% RSLogix 500 project Blue Banner Restacker.RSS, saved by version 11.00.00.00 %
PROJECT "UNTITLED"    % processor: MicroLogix 1400 %

PROGRAM FILES
  LAD 2   20 rungs

DATA FILES
  O0 OUTPUT  6 elements
  I1 INPUT  8 elements
  S2 STATUS  66 elements
  B3 BINARY  2 elements
  T4 TIMER  1 elements
  C5 COUNTER  1 elements
  R6 CONTROL  1 elements
  N7 INTEGER  1 elements
  F8 FLOAT  1 elements

LADDER 2
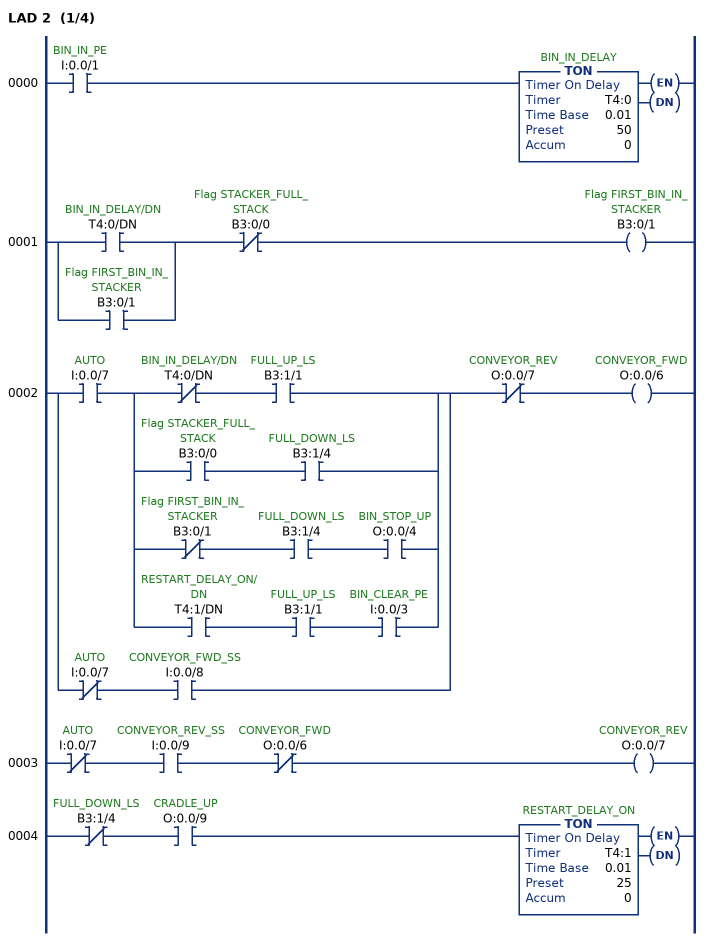
% Rung: 0 %  % edit flag set %
SOR XIC I:0.0/1 TON T4:0 0.01 50 0 EOR
%   I:0.0/1  BIN_IN_PE %
%   T4:0  BIN_IN_DELAY %
% Rung: 1 %  % edit flag set %
SOR BST XIC T4:0/DN NXB XIC B3:0/1 BND XIO B3:0/0 OTE B3:0/1 EOR
%   T4:0  BIN_IN_DELAY %
%   B3:0/1  FIRST_BIN_IN_STACKER  "Flag" %
%   B3:0/0  STACKER_FULL_STACK  "Flag" %
% Rung: 2 %  % edit flag set %
SOR BST XIC I:0.0/7 BST XIO T4:0/DN XIC B3:1/1 NXB BST XIC B3:0/0 XIC B3:1/4 NXB BST XIO B3:0/1 XIC B3:1/4 XIC O:0.0/4 NXB XIC T4:1/DN XIC B3:1/1 XIC I:0.0/3 BND BND BND NXB XIO I:0.0/7 XIC I:0.0/8 BND XIO O:0.0/7 OTE O:0.0/6 EOR
%   I:0.0/7  AUTO %
%   T4:0  BIN_IN_DELAY %
%   B3:1/1  FULL_UP_LS %
%   B3:0/0  STACKER_FULL_STACK  "Flag" %
%   B3:1/4  FULL_DOWN_LS %
%   B3:0/1  FIRST_BIN_IN_STACKER  "Flag" %
%   O:0.0/4  BIN_STOP_UP %
%   T4:1  RESTART_DELAY_ON %
%   I:0.0/3  BIN_CLEAR_PE %
%   I:0.0/8  CONVEYOR_FWD_SS %
%   O:0.0/7  CONVEYOR_REV %
%   O:0.0/6  CONVEYOR_FWD %
% Rung: 3 %  % edit flag set %
SOR XIO I:0.0/7 XIC I:0.0/9 XIO O:0.0/6 OTE O:0.0/7 EOR
%   I:0.0/7  AUTO %
%   I:0.0/9  CONVEYOR_REV_SS %
%   O:0.0/6  CONVEYOR_FWD %
%   O:0.0/7  CONVEYOR_REV %
% Rung: 4 %  % edit flag set %
SOR XIO B3:1/4 XIC O:0.0/9 TON T4:1 0.01 25 0 EOR
%   B3:1/4  FULL_DOWN_LS %
%   O:0.0/9  CRADLE_UP %
%   T4:1  RESTART_DELAY_ON %

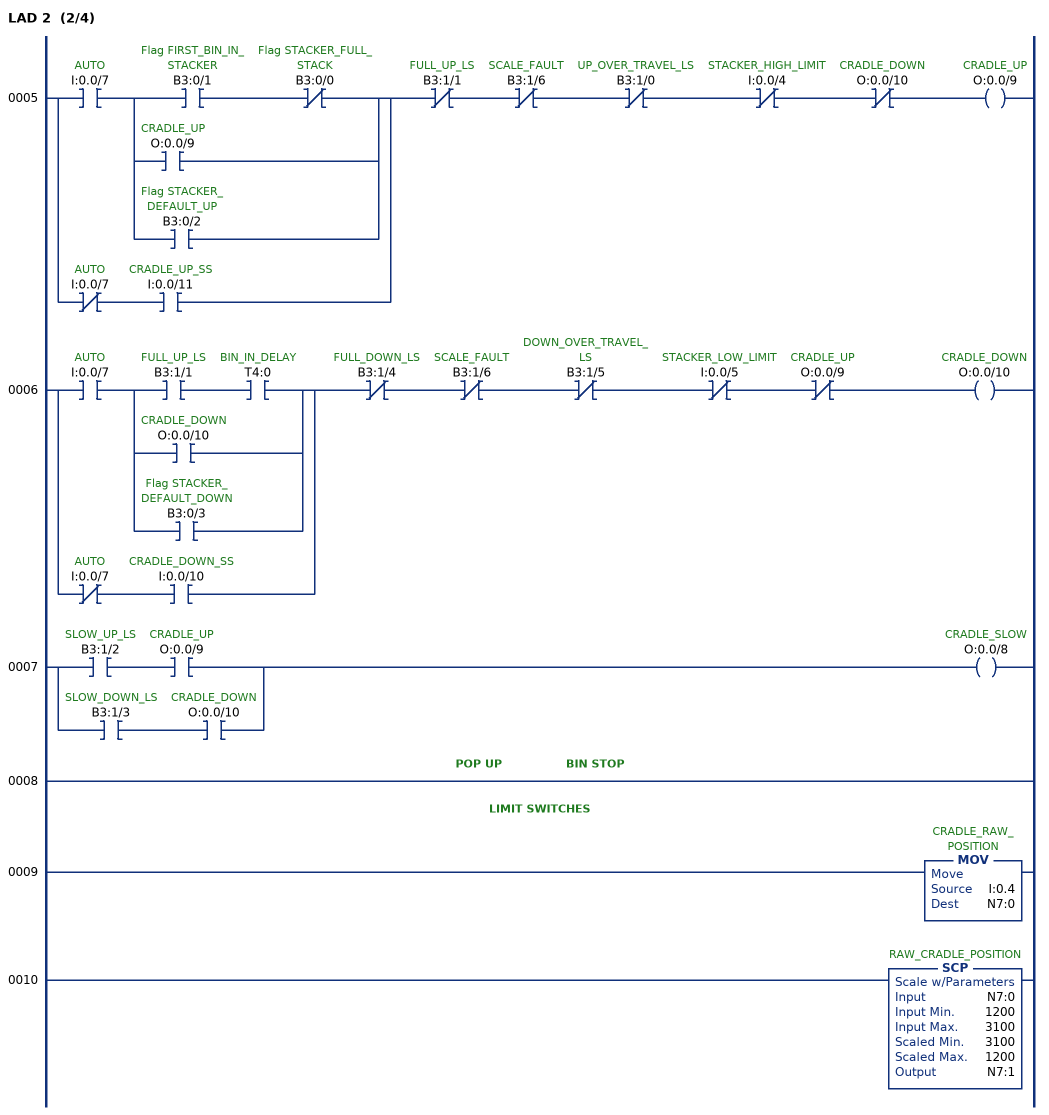
% Rung: 5 %  % edit flag set %
SOR BST XIC I:0.0/7 BST XIC B3:0/1 XIO B3:0/0 NXB BST XIC O:0.0/9 NXB XIC B3:0/2 BND BND NXB XIO I:0.0/7 XIC I:0.0/11 BND XIO B3:1/1 XIO B3:1/6 XIO B3:1/0 XIO I:0.0/4 XIO O:0.0/10 OTE O:0.0/9 EOR
%   I:0.0/7  AUTO %
%   B3:0/1  FIRST_BIN_IN_STACKER  "Flag" %
%   B3:0/0  STACKER_FULL_STACK  "Flag" %
%   O:0.0/9  CRADLE_UP %
%   B3:0/2  STACKER_DEFAULT_UP  "Flag" %
%   I:0.0/11  CRADLE_UP_SS %
%   B3:1/1  FULL_UP_LS %
%   B3:1/6  SCALE_FAULT %
%   B3:1/0  UP_OVER_TRAVEL_LS %
%   I:0.0/4  STACKER_HIGH_LIMIT %
%   O:0.0/10  CRADLE_DOWN %
% Rung: 6 %  % edit flag set %
SOR BST XIC I:0.0/7 BST XIC B3:1/1 XIC T4:0 NXB BST XIC O:0.0/10 NXB XIC B3:0/3 BND BND NXB XIO I:0.0/7 XIC I:0.0/10 BND XIO B3:1/4 XIO B3:1/6 XIO B3:1/5 XIO I:0.0/5 XIO O:0.0/9 OTE O:0.0/10 EOR
%   I:0.0/7  AUTO %
%   B3:1/1  FULL_UP_LS %
%   T4:0  BIN_IN_DELAY %
%   O:0.0/10  CRADLE_DOWN %
%   B3:0/3  STACKER_DEFAULT_DOWN  "Flag" %
%   I:0.0/10  CRADLE_DOWN_SS %
%   B3:1/4  FULL_DOWN_LS %
%   B3:1/6  SCALE_FAULT %
%   B3:1/5  DOWN_OVER_TRAVEL_LS %
%   I:0.0/5  STACKER_LOW_LIMIT %
%   O:0.0/9  CRADLE_UP %
% Rung: 7 %  % edit flag set %
SOR BST XIC B3:1/2 XIC O:0.0/9 NXB XIC B3:1/3 XIC O:0.0/10 BND OTE O:0.0/8 EOR
%   B3:1/2  SLOW_UP_LS %
%   O:0.0/9  CRADLE_UP %
%   B3:1/3  SLOW_DOWN_LS %
%   O:0.0/10  CRADLE_DOWN %
%   O:0.0/8  CRADLE_SLOW %
% Rung: 8 %  % edit flag set %
% TITLE: POP UP                BIN STOP %
SOR EOR
% Rung: 9 %  % edit flag set %
% TITLE: LIMIT SWITCHES %
SOR MOV I:0.4 N7:0 EOR
%   I:0.4  CRADLE_POSITION_RAW %
%   N7:0  CRADLE_RAW_POSITION %
% Rung: 10 %  % edit flag set %
SOR SCP N7:0 1200 3100 3100 1200 N7:1 EOR
%   N7:0  CRADLE_RAW_POSITION %
%   N7:1  RAW_CRADLE_POSITION %

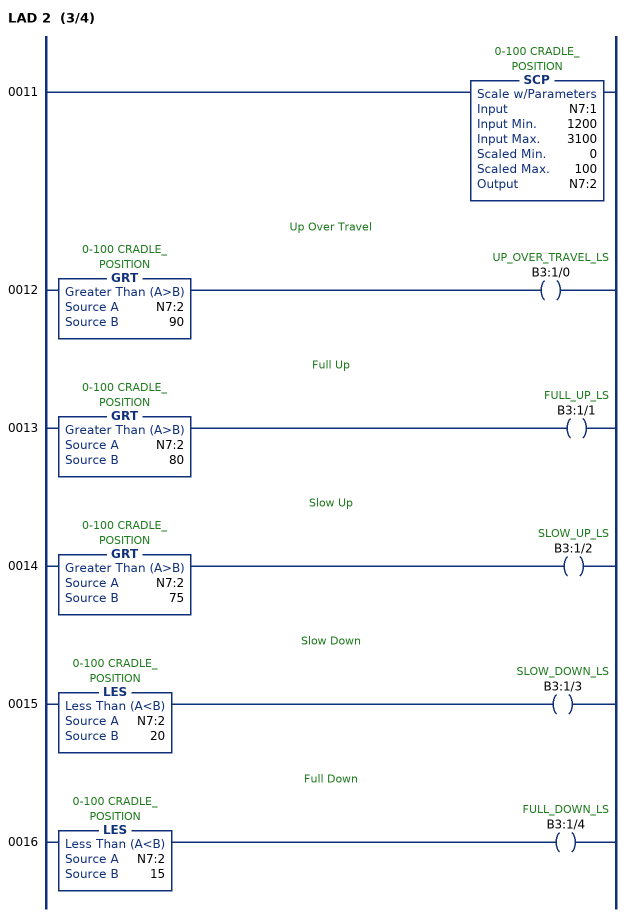
% Rung: 11 %  % edit flag set %
SOR SCP N7:1 1200 3100 0 100 N7:2 EOR
%   N7:1  RAW_CRADLE_POSITION %
%   N7:2  CRADLE_POSITION  "0-100" %
% Rung: 12 %  % edit flag set %
% Up Over Travel %
SOR GRT N7:2 90 OTE B3:1/0 EOR
%   N7:2  CRADLE_POSITION  "0-100" %
%   B3:1/0  UP_OVER_TRAVEL_LS %
% Rung: 13 %  % edit flag set %
% Full Up %
SOR GRT N7:2 80 OTE B3:1/1 EOR
%   N7:2  CRADLE_POSITION  "0-100" %
%   B3:1/1  FULL_UP_LS %
% Rung: 14 %  % edit flag set %
% Slow Up %
SOR GRT N7:2 75 OTE B3:1/2 EOR
%   N7:2  CRADLE_POSITION  "0-100" %
%   B3:1/2  SLOW_UP_LS %
% Rung: 15 %  % edit flag set %
% Slow Down %
SOR LES N7:2 20 OTE B3:1/3 EOR
%   N7:2  CRADLE_POSITION  "0-100" %
%   B3:1/3  SLOW_DOWN_LS %
% Rung: 16 %  % edit flag set %
% Full Down %
SOR LES N7:2 15 OTE B3:1/4 EOR
%   N7:2  CRADLE_POSITION  "0-100" %
%   B3:1/4  FULL_DOWN_LS %

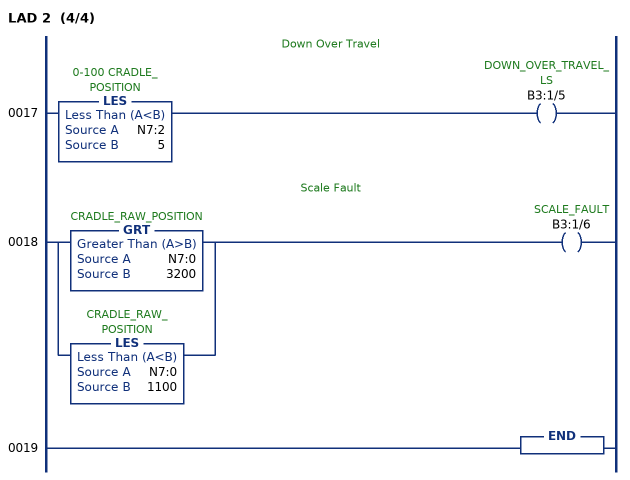
% Rung: 17 %  % edit flag set %
% Down Over Travel %
SOR LES N7:2 5 OTE B3:1/5 EOR
%   N7:2  CRADLE_POSITION  "0-100" %
%   B3:1/5  DOWN_OVER_TRAVEL_LS %
% Rung: 18 %  % edit flag set %
% Scale Fault %
SOR BST GRT N7:0 3200 NXB LES N7:0 1100 BND OTE B3:1/6 EOR
%   N7:0  CRADLE_RAW_POSITION %
%   B3:1/6  SCALE_FAULT %
% Rung: 19 %
SOR END EOR

OTHER DOCUMENTED ADDRESSES
  B3:5/2  "Stacker FULL Stack Flag"
  B3:5/3  "First Bin In Stacker Flag"
  B3:6/1  RESTACK_DOWN_LS
  B3:6/4  RESTACK_UP_LS
  I:0.0/0  BIN_APPROACH_PE
  I:0.0/2  FULL_STACK_PE
  I:0.0/12  BIN_STOP_UP_SS
  I:0.0/13  BIN_STOP_DOWN_SS
  I:0.0/15  STACKER_RUNNING_MO1
  I:0.1/3  LS4  "Outfeed Barrier/Unstacker StageLS"
  I:2.0/0  MANUAL_RESTACK_FWD  "SEL_RESTACK_CONV_FWD"
  I:2.0/11  PE10  "Pop up conv stage PE"
  O:0.0/1  RUN
  O:0.0/5  BIN_STOP_DOWN
  O:3.0/5  RESTACKER_UP
  O:5.0/4  RESTACKER_CONV_FWD  "Restacker Conv FWD"
  O:5.0/14  RESTACK_BIN_STOP_UP
  O:5.0/15  STACK_UNLOAD_POP_UP  "pop up conveyor"
  T4:50/TT  P
